Yaskawa INFORM job: valve_cylinder_program.JBI

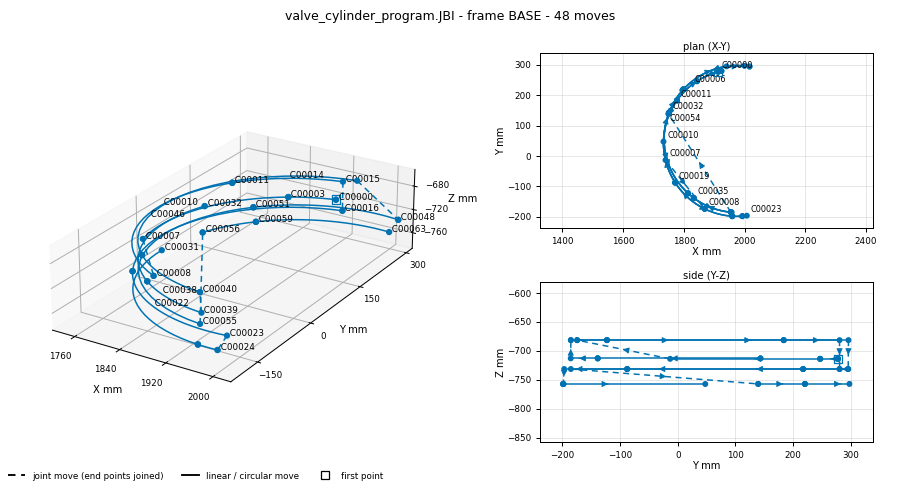
[picture p0: tool path of valve_cylinder_program.JBI in frame BASE, 48 of 69 moves have a stored position in this frame; points joined in program order, loops and branches not executed]
/JOB
//NAME valve_cylinder_program
//POS
///NPOS 64,0,64,0,0,0
///TOOL 0
///POSTYPE BASE
///RECTAN
///RCONF 0,0,0,0,0,0,0,0,0,0,0,0,0,0,0,0,0,0,0,0,0,0,0,0
C00000=1912.956375,277.467732,-713.734000,104.845113,-90.000000,5.000000
C00001=1912.956375,277.467732,-713.734000,104.845113,-90.000000,5.000000
C00002=1875.741540,264.271552,-713.734000,114.203351,-90.000000,5.000000
C00003=1843.232351,246.554196,-713.734000,122.977004,-90.000000,5.000000
C00004=1843.232351,246.554196,-713.734000,122.977004,-90.000000,5.000000
C00005=1843.232351,246.554196,-713.734000,122.977004,-90.000000,5.000000
C00006=1821.867134,230.969302,-713.734000,129.240888,-89.999999,5.000000
C00007=1739.660322,-13.084066,-713.734000,-166.472003,-90.000000,5.000000
C00008=1868.777508,-173.949937,-681.434960,175.000000,-60.000000,63.975761
C00009=1868.777508,-173.949937,-681.434960,175.000000,-60.000000,63.975761
C00010=1732.977573,47.454213,-681.434960,175.000000,-60.000000,-5.000000
C00011=1777.446525,183.384272,-681.434960,-175.000000,-60.000000,-35.301206
C00012=1777.446525,183.384272,-681.434960,-175.000000,-60.000000,-35.301206
C00013=1777.446525,183.384272,-681.434960,-175.000000,-60.000000,-35.301206
C00014=1841.519513,245.432520,-681.434960,175.000000,-60.000000,-56.538281
C00015=1923.540673,280.019785,-681.434960,175.000000,-60.000000,-77.732669
C00016=1923.679580,280.049946,-731.362460,175.000000,-60.000000,-77.766320
C00017=1923.679580,280.049946,-731.362460,175.000000,-60.000000,-77.766320
C00018=1733.926305,21.764774,-731.362460,175.000000,-60.000000,5.159418
C00019=1771.436507,-87.426687,-731.362460,175.000000,-60.000000,32.758531
C00020=1771.436507,-87.426687,-731.362460,175.000000,-60.000000,32.758531
C00021=1771.436507,-87.426687,-731.362460,175.000000,-60.000000,32.758531
C00022=1863.629238,-171.359902,-731.362460,175.000000,-60.000000,62.611364
C00023=2007.406066,-196.303988,-731.362460,-175.000000,-60.000000,97.703890
C00024=1992.473798,-197.854083,-757.277960,175.000000,-60.000000,94.149218
C00025=1992.473798,-197.854083,-757.277960,175.000000,-60.000000,94.149218
C00026=1973.279386,-198.482555,-757.277960,-175.000000,-60.000000,89.601453
C00027=1959.496793,-197.993728,-757.277960,-175.000000,-60.000000,86.336031
C00028=1959.496793,-197.993728,-757.277960,-175.000000,-60.000000,86.336031
C00029=1959.496793,-197.993728,-757.277960,-175.000000,-60.000000,86.336031
C00030=1735.068001,11.548301,-757.277960,175.000000,-60.000000,7.593332
C00031=1732.981838,47.708853,-757.277960,175.000000,-60.000000,-5.000000
C00032=1751.144686,143.223321,-712.914500,158.917483,-89.999999,5.000000
C00033=1751.144686,143.223321,-712.914500,158.917483,-89.999999,5.000000
C00034=1807.656401,-116.772170,-712.914500,-134.391742,-89.999999,5.000000
C00035=1832.924507,-138.320913,-712.914500,-126.523616,-90.000000,5.000000
C00036=1832.924507,-138.320913,-712.914500,-126.523616,-90.000000,5.000000
C00037=1832.924507,-138.320913,-712.914500,-126.523616,-90.000000,5.000000
C00038=1870.260183,-161.058862,-712.914500,-116.160382,-90.000000,5.000000
C00039=1957.474949,-185.064445,-712.914500,-94.618409,-90.000000,5.000000
C00040=1955.066601,-184.857785,-681.396960,175.000000,-60.000000,84.809334
C00041=1955.066601,-184.857785,-681.396960,175.000000,-60.000000,84.809334
C00042=1902.518613,-174.116602,-681.396960,175.000000,-60.000000,72.085620
C00043=1813.615063,-122.411056,-681.396960,-175.000000,-60.000000,47.550546
C00044=1813.615063,-122.411056,-681.396960,-175.000000,-60.000000,47.550546
C00045=1813.615063,-122.411056,-681.396960,-175.000000,-60.000000,47.550546
C00046=1741.393691,0.670328,-681.396960,-175.000000,-60.000000,13.256347
C00047=1940.755973,295.460388,-681.396960,175.000000,-60.000000,-81.396196
C00048=2016.389804,294.950680,-731.369960,175.000000,-60.000000,-99.376042
C00049=2016.389804,294.950680,-731.369960,175.000000,-60.000000,-99.376042
C00050=1893.660369,283.396063,-731.369960,-175.000000,-60.000000,-69.867204
C00051=1796.087616,216.967166,-731.369960,175.000000,-60.000000,-41.637631
C00052=1796.087616,216.967166,-731.369960,175.000000,-60.000000,-41.637631
C00053=1796.087616,216.967166,-731.369960,175.000000,-60.000000,-41.637631
C00054=1739.832762,104.561215,-731.369960,175.000000,-60.000000,-11.534774
C00055=1954.877451,-184.840527,-731.369960,175.000000,-60.000000,84.764368
C00056=1749.641928,139.220287,-757.137960,175.000000,-60.000000,-20.070237
C00057=1749.641928,139.220287,-757.137960,175.000000,-60.000000,-20.070237
C00058=1774.832702,189.268439,-757.137960,175.000000,-60.000000,-33.364800
C00059=1798.921286,220.099117,-757.137960,175.000000,-60.000000,-42.637550
C00060=1798.921286,220.099117,-757.137960,175.000000,-60.000000,-42.637550
C00061=1798.921286,220.099117,-757.137960,175.000000,-60.000000,-42.637550
C00062=1837.803510,254.174919,-757.137960,-175.000000,-60.000000,-54.900765
C00063=1999.627377,297.120271,-757.137960,175.000000,-60.000000,-95.373744
///POSTYPE PULSE
///PULSE
EX00000=102400.0
EX00001=269312.0
///POSTYPE PULSE
///PULSE
EC00000=102400.0
EC00001=102400.0
EC00002=102400.0
EC00003=102400.0
EC00004=102400.0
EC00005=102400.0
EC00006=102400.0
EC00007=102400.0
EC00008=102400.0
EC00009=102400.0
EC00010=102400.0
EC00011=102400.0
EC00012=102400.0
EC00013=102400.0
EC00014=102400.0
EC00015=102400.0
EC00016=102400.0
EC00017=102400.0
EC00018=102400.0
EC00019=102400.0
EC00020=102400.0
EC00021=102400.0
EC00022=102400.0
EC00023=102400.0
EC00024=102400.0
EC00025=102400.0
EC00026=102400.0
EC00027=102400.0
EC00028=102400.0
EC00029=102400.0
EC00030=102400.0
EC00031=102400.0
EC00032=269312.0
EC00033=269312.0
EC00034=269312.0
EC00035=269312.0
EC00036=269312.0
EC00037=269312.0
EC00038=269312.0
EC00039=269312.0
EC00040=269312.0
EC00041=269312.0
EC00042=269312.0
EC00043=269312.0
EC00044=269312.0
EC00045=269312.0
EC00046=269312.0
EC00047=269312.0
EC00048=269312.0
EC00049=269312.0
EC00050=269312.0
EC00051=269312.0
EC00052=269312.0
EC00053=269312.0
EC00054=269312.0
EC00055=269312.0
EC00056=269312.0
EC00057=269312.0
EC00058=269312.0
EC00059=269312.0
EC00060=269312.0
EC00061=269312.0
EC00062=269312.0
EC00063=269312.0
//INST
///DATE 2023/08/16 18:06
///ATTR SC,RW,RJ
////FRAME BASE
///GROUP1 RB1,ST1
NOP
MOVJ P009 EX000 VJ=15.00
MOVJ C00000 EC00000 VJ=15.0
CALL JOB:SPYON
MOVC C00001 EC00001 V=150.0
MOVC C00002 EC00002 V=150.0
MOVC C00003 EC00003 V=150.0
MOVJ C00004 EC00004 VJ=15.0
MOVC C00005 EC00005 V=150.0
MOVC C00006 EC00006 V=150.0
MOVC C00007 EC00007 V=150.0
MOVJ C00008 EC00008 VJ=15.0
MOVC C00009 EC00009 V=150.0
MOVC C00010 EC00010 V=150.0
MOVC C00011 EC00011 V=150.0
MOVJ C00012 EC00012 VJ=15.0
MOVC C00013 EC00013 V=150.0
MOVC C00014 EC00014 V=150.0
MOVC C00015 EC00015 V=150.0
MOVJ C00016 EC00016 VJ=15.0
MOVC C00017 EC00017 V=150.0
MOVC C00018 EC00018 V=150.0
MOVC C00019 EC00019 V=150.0
MOVJ C00020 EC00020 VJ=15.0
MOVC C00021 EC00021 V=150.0
MOVC C00022 EC00022 V=150.0
MOVC C00023 EC00023 V=150.0
MOVJ C00024 EC00024 VJ=15.0
MOVC C00025 EC00025 V=150.0
MOVC C00026 EC00026 V=150.0
MOVC C00027 EC00027 V=150.0
MOVJ C00028 EC00028 VJ=15.0
MOVC C00029 EC00029 V=150.0
MOVC C00030 EC00030 V=150.0
MOVC C00031 EC00031 V=150.0
CALL JOB:SPYOF
MOVJ P009 VJ=15.00
MOVL P009 EX00000 V=150.0
MOVJ C00032 EC00032 VJ=15.0
CALL JOB:SPYON
MOVC C00033 EC00033 V=150.0
MOVC C00034 EC00034 V=150.0
MOVC C00035 EC00035 V=150.0
MOVJ C00036 EC00036 VJ=15.0
MOVC C00037 EC00037 V=150.0
MOVC C00038 EC00038 V=150.0
MOVC C00039 EC00039 V=150.0
MOVJ C00040 EC00040 VJ=15.0
MOVC C00041 EC00041 V=150.0
MOVC C00042 EC00042 V=150.0
MOVC C00043 EC00043 V=150.0
MOVJ C00044 EC00044 VJ=15.0
MOVC C00045 EC00045 V=150.0
MOVC C00046 EC00046 V=150.0
MOVC C00047 EC00047 V=150.0
MOVJ C00048 EC00048 VJ=15.0
MOVC C00049 EC00049 V=150.0
MOVC C00050 EC00050 V=150.0
MOVC C00051 EC00051 V=150.0
MOVJ C00052 EC00052 VJ=15.0
MOVC C00053 EC00053 V=150.0
MOVC C00054 EC00054 V=150.0
MOVC C00055 EC00055 V=150.0
MOVJ C00056 EC00056 VJ=15.0
MOVC C00057 EC00057 V=150.0
MOVC C00058 EC00058 V=150.0
MOVC C00059 EC00059 V=150.0
MOVJ C00060 EC00060 VJ=15.0
MOVC C00061 EC00061 V=150.0
MOVC C00062 EC00062 V=150.0
MOVC C00063 EC00063 V=150.0
CALL JOB:SPYOF
MOVJ P009 VJ=15.00
MOVL P009 EX00001 V=150.0
END
